FUNCTION F_CalcValuesHeatSteam : REAL
VAR_INPUT
	rTempFinal		: REAL;				// [°C]		
	rTempInitial	: REAL;				// [°C]		
	rCT				: REAL;				// []		Coefficient for temperature
	rCS				: REAL;				// []		Coefficient for steam
	rCA				: REAL;				// []		Coefficient for airflow
	rMachineLength	: REAL;				// [m]		Length of machine
	// Limits
	rTimeMin		: REAL;				// [s]		Minimum allowed time in machine
	rTimeMax		: REAL;				// [s]		Maximum allowed time in machine
	rTempMin		: REAL;				// [°C]		Minimum allowed temperature in machine
	rTempMax		: REAL;				// [°C]		Maximum allowed temperature in machine
	rSteamMin		: REAL;				// []		Minimum allowed steam in machine
	rSteamMax		: REAL;				// []		Maximum allowed steam in machine
	rAirMin			: REAL;				// []		Minimum allowed airflow in machine
	rAirMax			: REAL;				// []		Maximum allowed airflow in machine	
END_VAR
VAR_OUTPUT
	rVelocity		: REAL;				// [m/s]	Carrier velocity
	rTempMachine	: REAL;				// [°C]		Machine temperature
	rTimeMachine	: REAL;				// [s]		Time in machine
	rSteamMachine	: REAL;				// []		
	rAirMachine		: REAL;				// []		
END_VAR
VAR
	// Limits
	rVelocityMin	: REAL := 0.001;	// [m/s]	Minimum allowed speed
	rVelocityMax	: REAL := 2.0;		// [m/s]	Maximum allowed speed
	
	// Temp
	rVelocityCalcRaw: REAL;				// [m/s]	
	rVelocityCalc	: REAL;				// [m/s]	
	rTimeCalcRaw	: REAL;				// [s]		
	rTimeCalc		: REAL;				// [s]		
	sTempString		: STRING(200);		// 			
END_VAR


// Calculate time needed in device and machine temperature
//t = ( (TFinal) / (TMachine * cT + SMachine * cS + AMachine * cA) ) - TInitial

// If constants are ZERO use fixed time in mechine from job data (minimum time)
IF ( (rCT = 0.0) AND (rCS = 0.0) AND (rCA = 0.0) ) THEN
	rTimeCalcRaw := rTimeMin;
	rTempMachine := rTempMax;
	rSteamMachine := rSteamMax;
	rAirMax := rAirMax;
	
ELSE
	rTempMachine := (rTempMin + rTempMax) / 2.0;
	rSteamMachine := (rSteamMin + rSteamMax) / 2.0;
	rAirMachine := (rAirMin + rAirMax) / 2.0;

	// Check for divide-by-zero
	IF ((rTempMachine * rCT) + (rSteamMachine * rCS) + (rAirMachine * rCA)) = 0.0 THEN
		rTimeCalcRaw := rTimeMin;
		rTempMachine := rTempMax;
		rSteamMachine := rSteamMax;
		rAirMax := rAirMax;
	ELSE
		rTimeCalcRaw := (rTempFinal - rTempInitial) / ((rTempMachine * rCT) + (rSteamMachine * rCS) + (rAirMachine * rCA));	
	END_IF
	
END_IF

// Limit time in device according to job data
rTimeCalc := LIMIT(rTimeMin, rTimeCalcRaw, rTimeMax);

// Make sure time is not ZERO
IF (rTimeCalc <= 0.0) THEN
	rTimeCalc := 120.0;

END_IF

// Calculate velocity based on time in machine and machine length
rVelocityCalcRaw := rMachineLength / rTimeCalc;

// Limit velocity to allowed limits
rVelocityCalc := LIMIT(rVelocityMin, rVelocityCalcRaw, rVelocityMax);

// Log
	sTempString := CONCAT('STAT: ', 'Velocity Calc ');
	sTempString := CONCAT(sTempString, '. Temp=');
	sTempString := CONCAT(sTempString, TO_STRING(rTempMachine));
	sTempString := CONCAT(sTempString, '. Steam=');
	sTempString := CONCAT(sTempString, TO_STRING(rSteamMachine));
	sTempString := CONCAT(sTempString, '. Air=');
	sTempString := CONCAT(sTempString, TO_STRING(rAirMachine));
	sTempString := CONCAT(sTempString, '. Time_RAW=');
	sTempString := CONCAT(sTempString, TO_STRING(rTimeCalcRaw));
	sTempString := CONCAT(sTempString, '. Time=');
	sTempString := CONCAT(sTempString, TO_STRING(rTimeCalc));
	sTempString := CONCAT(sTempString, '. Vel_RAW=');
	sTempString := CONCAT(sTempString, TO_STRING(rVelocityCalcRaw));
	sTempString := CONCAT(sTempString, '. Vel=');
	sTempString := CONCAT(sTempString, TO_STRING(rVelocityCalc));
	F_Logfile(sTempString);

// Output
rVelocity := rVelocityCalc;
rTempMachine := rTempMachine;
rSteamMachine := rSteamMachine;
rAirMachine := rAirMachine;
rTimeMachine := rTimeCalc;

END_FUNCTION

(* stored: Version 1.1.0.1, ProductVersion 3.1.4024.5
   POU F_CalcValuesHeatSteam: Id {99f54be2-3f5d-4397-b7f4-3cbaaee12bb6}, SpecialFunc None *)
